TYPE ST_Frequency :
STRUCT
	Frequency:	REAL;
END_STRUCT
END_TYPE

(* stored: Version 1.1.0.1, ProductVersion 3.1.4020.6
   DUT ST_Frequency: Id {eee7e4e4-e6d9-4646-b9e1-1365a7280519} *)
